PROGRAM RunGRAB
VAR

END_VAR
VAR CONSTANT 
    HOMING: INT := 1;
	MANUAL: INT := 2;
	POSITION: INT := 3;
	STOP: INT := 4;
END_VAR

// State machine
CASE GVL.stateGRAB OF
HOMING:
	.Homing();
	
MANUAL:
	.ManualHorAxis();
	.ManualRotAxis();
	
POSITION:
	.PositionHorAxis();
	.PositionRotAxis();
	
STOP:
	//SAMELUR

ELSE
	// GRAB waiting for command
END_CASE

END_PROGRAM

(* stored: Version 1.1.0.1, ProductVersion 3.1.4024.6
   POU RunGRAB: Id {197f5f68-78b2-4da9-9af1-69511c5d94d2}, SpecialFunc None *)
